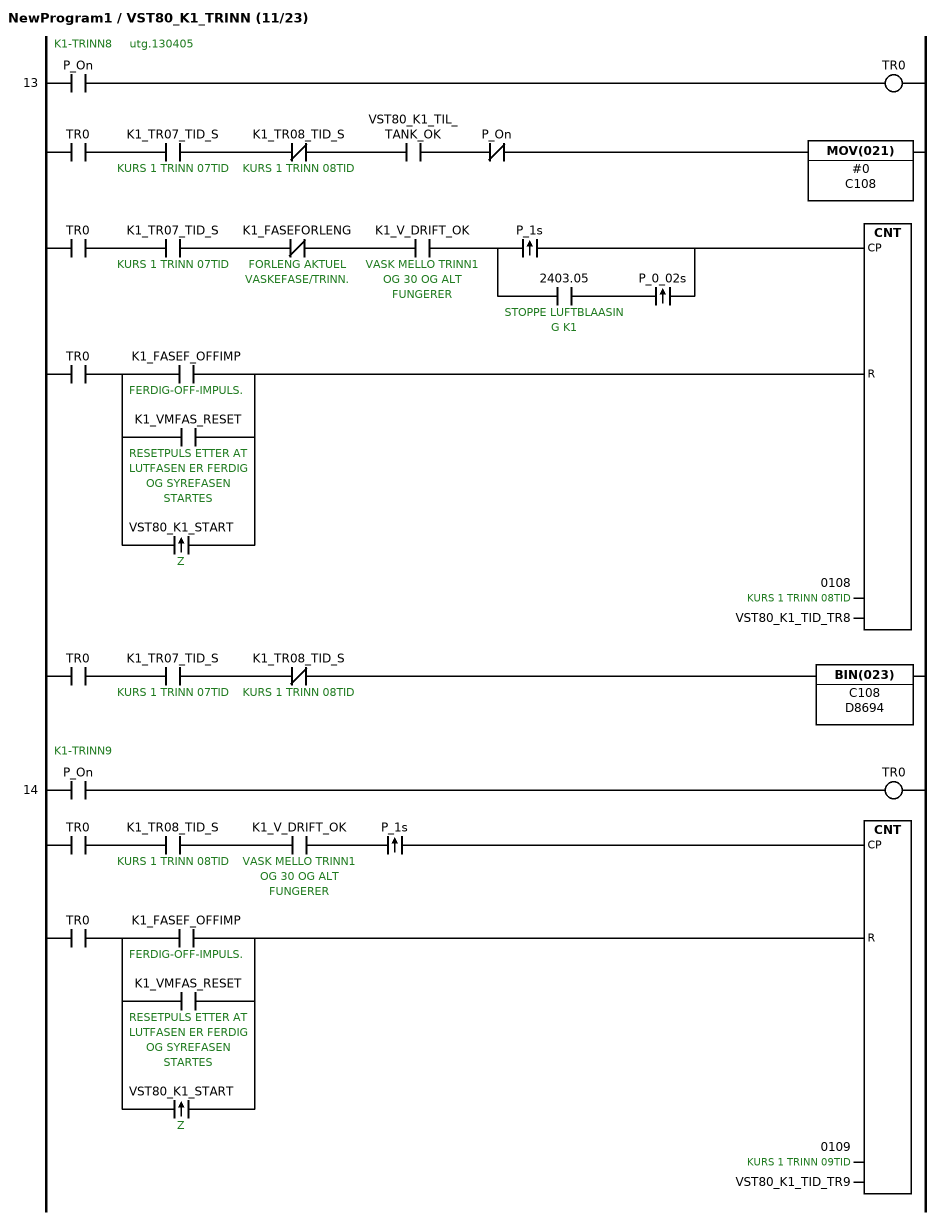
; [picture p96: NewProgram1 / VST80_K1_TRINN, rungs 13-14]
; rung 13: K1-TRINN8     utg.130405
LD P_On
OUT TR0
AND K1_TR07_TID_S  ; KURS 1 TRINN 07TID
ANDNOT K1_TR08_TID_S  ; KURS 1 TRINN 08TID
AND VST80_K1_TIL_TANK_OK
ANDNOT P_On
MOV(021) #0 C108
LD TR0
AND K1_TR07_TID_S  ; KURS 1 TRINN 07TID
ANDNOT K1_FASEFORLENG  ; FORLENG AKTUEL VASKEFASE/TRINN.
AND K1_V_DRIFT_OK  ; VASK MELLO TRINN1 OG 30 OG ALT FUNGERER
@LD P_1s
LD 2403.05  ; STOPPE LUFTBLAASING K1
@AND P_0_02s
ORLD
ANDLD
LD TR0
LD K1_FASEF_OFFIMP  ; FERDIG-OFF-IMPULS.
OR K1_VMFAS_RESET  ; RESETPULS ETTER AT LUTFASEN ER FERDIG OG SYREFASEN STARTES
@OR VST80_K1_START  ; Z
ANDLD
CNT 0108 VST80_K1_TID_TR8  ; KURS 1 TRINN 08TID
LD TR0
AND K1_TR07_TID_S  ; KURS 1 TRINN 07TID
ANDNOT K1_TR08_TID_S  ; KURS 1 TRINN 08TID
BIN(023) C108 D8694
; rung 14: K1-TRINN9
LD P_On
OUT TR0
AND K1_TR08_TID_S  ; KURS 1 TRINN 08TID
AND K1_V_DRIFT_OK  ; VASK MELLO TRINN1 OG 30 OG ALT FUNGERER
@AND P_1s
LD TR0
LD K1_FASEF_OFFIMP  ; FERDIG-OFF-IMPULS.
OR K1_VMFAS_RESET  ; RESETPULS ETTER AT LUTFASEN ER FERDIG OG SYREFASEN STARTES
@OR VST80_K1_START  ; Z
ANDLD
CNT 0109 VST80_K1_TID_TR9  ; KURS 1 TRINN 09TID

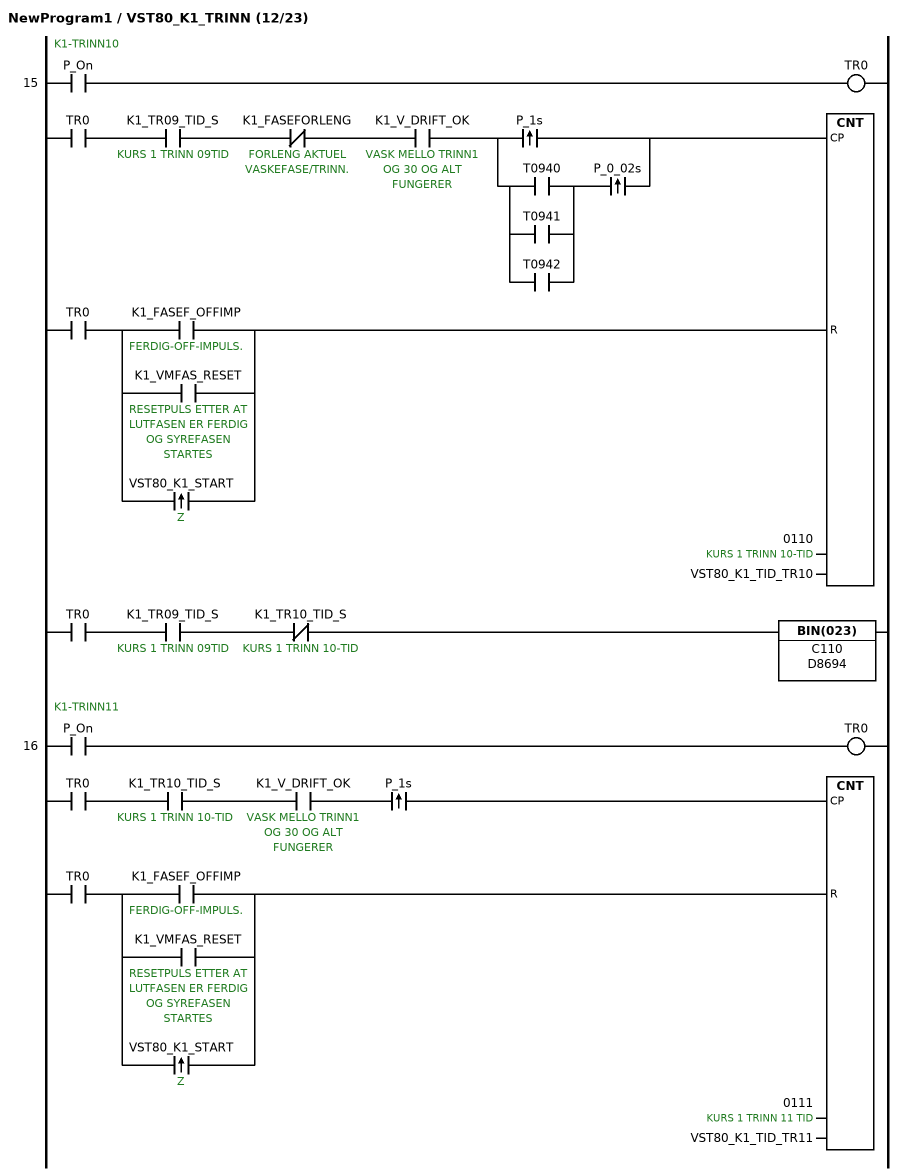
; rung 15: K1-TRINN10
LD P_On
OUT TR0
AND K1_TR09_TID_S  ; KURS 1 TRINN 09TID
ANDNOT K1_FASEFORLENG  ; FORLENG AKTUEL VASKEFASE/TRINN.
AND K1_V_DRIFT_OK  ; VASK MELLO TRINN1 OG 30 OG ALT FUNGERER
@LD P_1s
LD T0940
OR T0941
OR T0942
@AND P_0_02s
ORLD
ANDLD
LD TR0
LD K1_FASEF_OFFIMP  ; FERDIG-OFF-IMPULS.
OR K1_VMFAS_RESET  ; RESETPULS ETTER AT LUTFASEN ER FERDIG OG SYREFASEN STARTES
@OR VST80_K1_START  ; Z
ANDLD
CNT 0110 VST80_K1_TID_TR10  ; KURS 1 TRINN 10-TID
LD TR0
AND K1_TR09_TID_S  ; KURS 1 TRINN 09TID
ANDNOT K1_TR10_TID_S  ; KURS 1 TRINN 10-TID
BIN(023) C110 D8694
; rung 16: K1-TRINN11
LD P_On
OUT TR0
AND K1_TR10_TID_S  ; KURS 1 TRINN 10-TID
AND K1_V_DRIFT_OK  ; VASK MELLO TRINN1 OG 30 OG ALT FUNGERER
@AND P_1s
LD TR0
LD K1_FASEF_OFFIMP  ; FERDIG-OFF-IMPULS.
OR K1_VMFAS_RESET  ; RESETPULS ETTER AT LUTFASEN ER FERDIG OG SYREFASEN STARTES
@OR VST80_K1_START  ; Z
ANDLD
CNT 0111 VST80_K1_TID_TR11  ; KURS 1 TRINN 11 TID

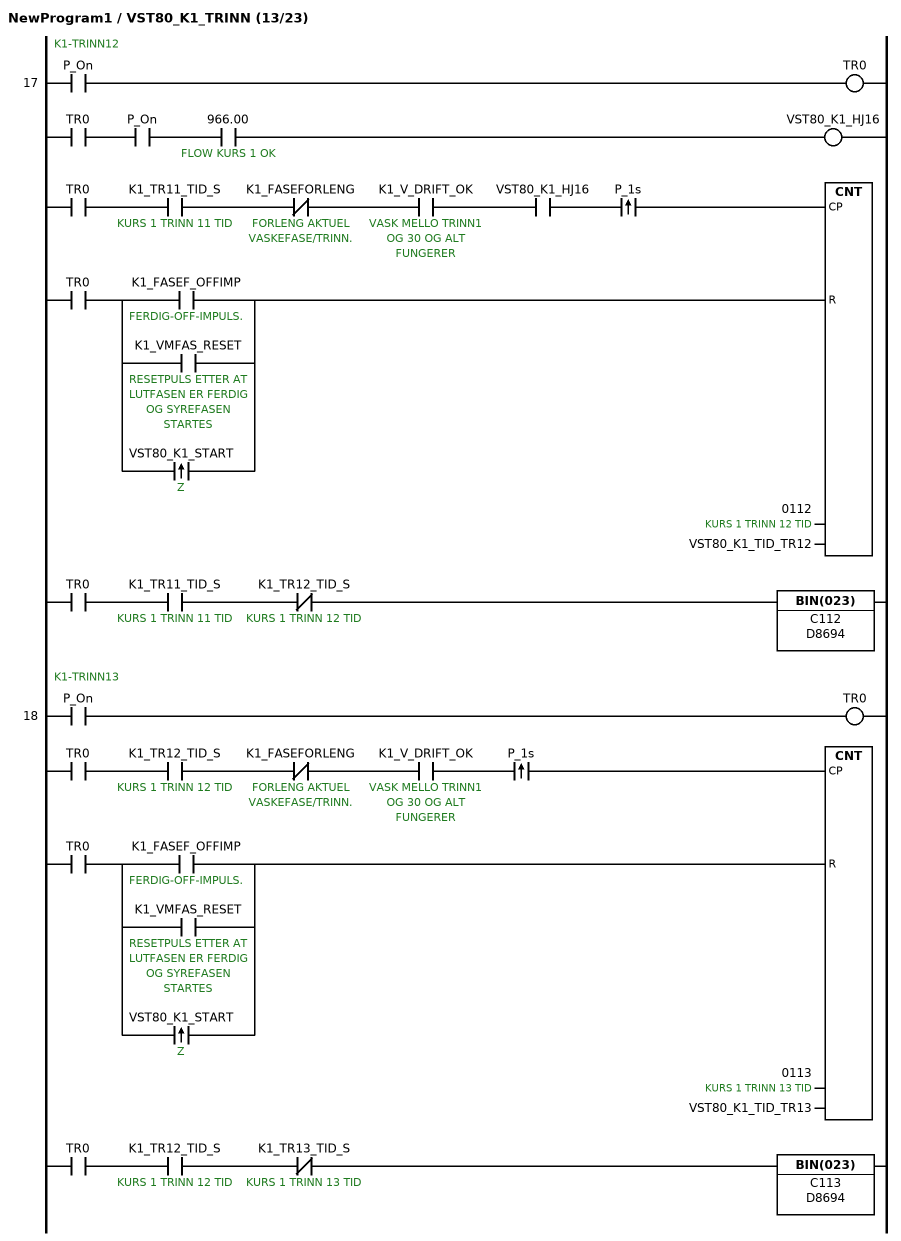
; rung 17: K1-TRINN12
LD P_On
OUT TR0
AND P_On
AND 966.00  ; FLOW KURS 1 OK
OUT VST80_K1_HJ16
LD TR0
AND K1_TR11_TID_S  ; KURS 1 TRINN 11 TID
ANDNOT K1_FASEFORLENG  ; FORLENG AKTUEL VASKEFASE/TRINN.
AND K1_V_DRIFT_OK  ; VASK MELLO TRINN1 OG 30 OG ALT FUNGERER
AND VST80_K1_HJ16
@AND P_1s
LD TR0
LD K1_FASEF_OFFIMP  ; FERDIG-OFF-IMPULS.
OR K1_VMFAS_RESET  ; RESETPULS ETTER AT LUTFASEN ER FERDIG OG SYREFASEN STARTES
@OR VST80_K1_START  ; Z
ANDLD
CNT 0112 VST80_K1_TID_TR12  ; KURS 1 TRINN 12 TID
LD TR0
AND K1_TR11_TID_S  ; KURS 1 TRINN 11 TID
ANDNOT K1_TR12_TID_S  ; KURS 1 TRINN 12 TID
BIN(023) C112 D8694
; rung 18: K1-TRINN13
LD P_On
OUT TR0
AND K1_TR12_TID_S  ; KURS 1 TRINN 12 TID
ANDNOT K1_FASEFORLENG  ; FORLENG AKTUEL VASKEFASE/TRINN.
AND K1_V_DRIFT_OK  ; VASK MELLO TRINN1 OG 30 OG ALT FUNGERER
@AND P_1s
LD TR0
LD K1_FASEF_OFFIMP  ; FERDIG-OFF-IMPULS.
OR K1_VMFAS_RESET  ; RESETPULS ETTER AT LUTFASEN ER FERDIG OG SYREFASEN STARTES
@OR VST80_K1_START  ; Z
ANDLD
CNT 0113 VST80_K1_TID_TR13  ; KURS 1 TRINN 13 TID
LD TR0
AND K1_TR12_TID_S  ; KURS 1 TRINN 12 TID
ANDNOT K1_TR13_TID_S  ; KURS 1 TRINN 13 TID
BIN(023) C113 D8694

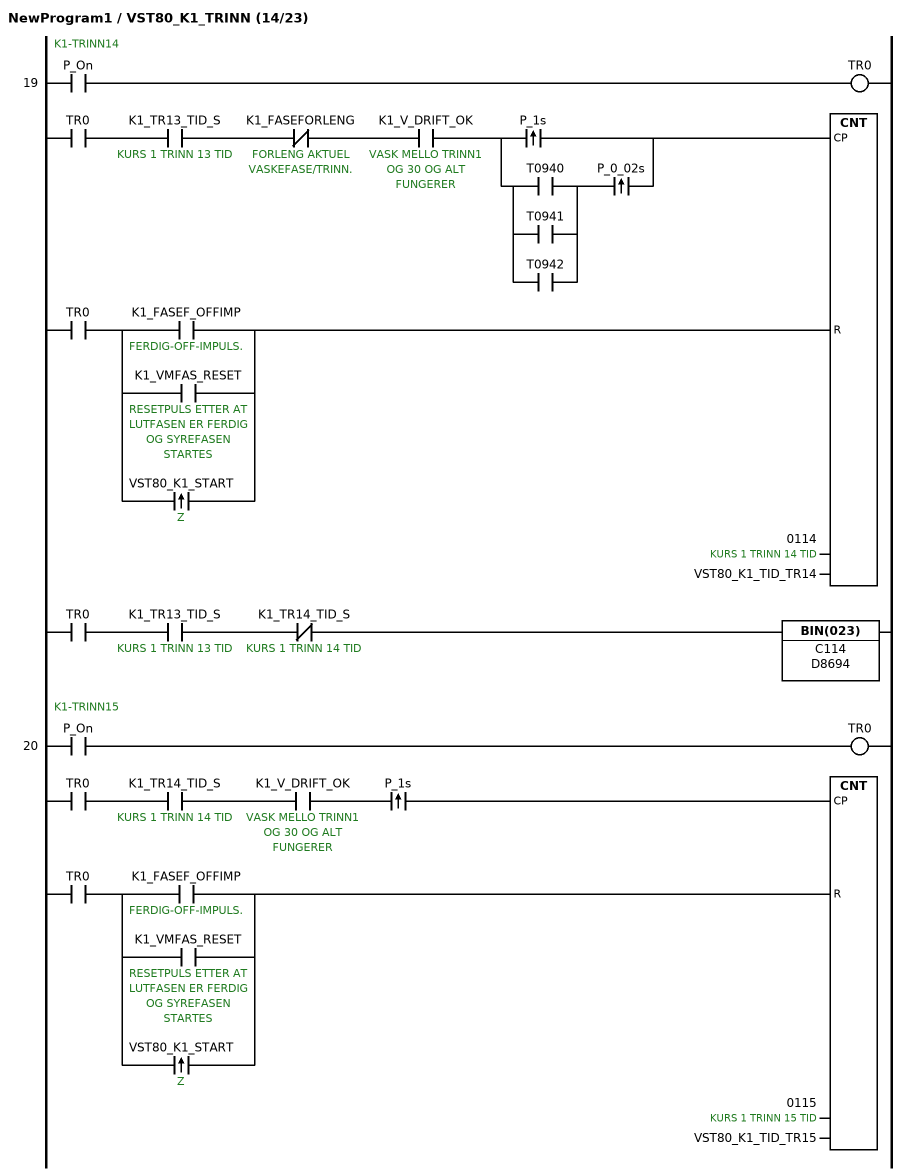
; rung 19: K1-TRINN14
LD P_On
OUT TR0
AND K1_TR13_TID_S  ; KURS 1 TRINN 13 TID
ANDNOT K1_FASEFORLENG  ; FORLENG AKTUEL VASKEFASE/TRINN.
AND K1_V_DRIFT_OK  ; VASK MELLO TRINN1 OG 30 OG ALT FUNGERER
@LD P_1s
LD T0940
OR T0941
OR T0942
@AND P_0_02s
ORLD
ANDLD
LD TR0
LD K1_FASEF_OFFIMP  ; FERDIG-OFF-IMPULS.
OR K1_VMFAS_RESET  ; RESETPULS ETTER AT LUTFASEN ER FERDIG OG SYREFASEN STARTES
@OR VST80_K1_START  ; Z
ANDLD
CNT 0114 VST80_K1_TID_TR14  ; KURS 1 TRINN 14 TID
LD TR0
AND K1_TR13_TID_S  ; KURS 1 TRINN 13 TID
ANDNOT K1_TR14_TID_S  ; KURS 1 TRINN 14 TID
BIN(023) C114 D8694
; rung 20: K1-TRINN15
LD P_On
OUT TR0
AND K1_TR14_TID_S  ; KURS 1 TRINN 14 TID
AND K1_V_DRIFT_OK  ; VASK MELLO TRINN1 OG 30 OG ALT FUNGERER
@AND P_1s
LD TR0
LD K1_FASEF_OFFIMP  ; FERDIG-OFF-IMPULS.
OR K1_VMFAS_RESET  ; RESETPULS ETTER AT LUTFASEN ER FERDIG OG SYREFASEN STARTES
@OR VST80_K1_START  ; Z
ANDLD
CNT 0115 VST80_K1_TID_TR15  ; KURS 1 TRINN 15 TID

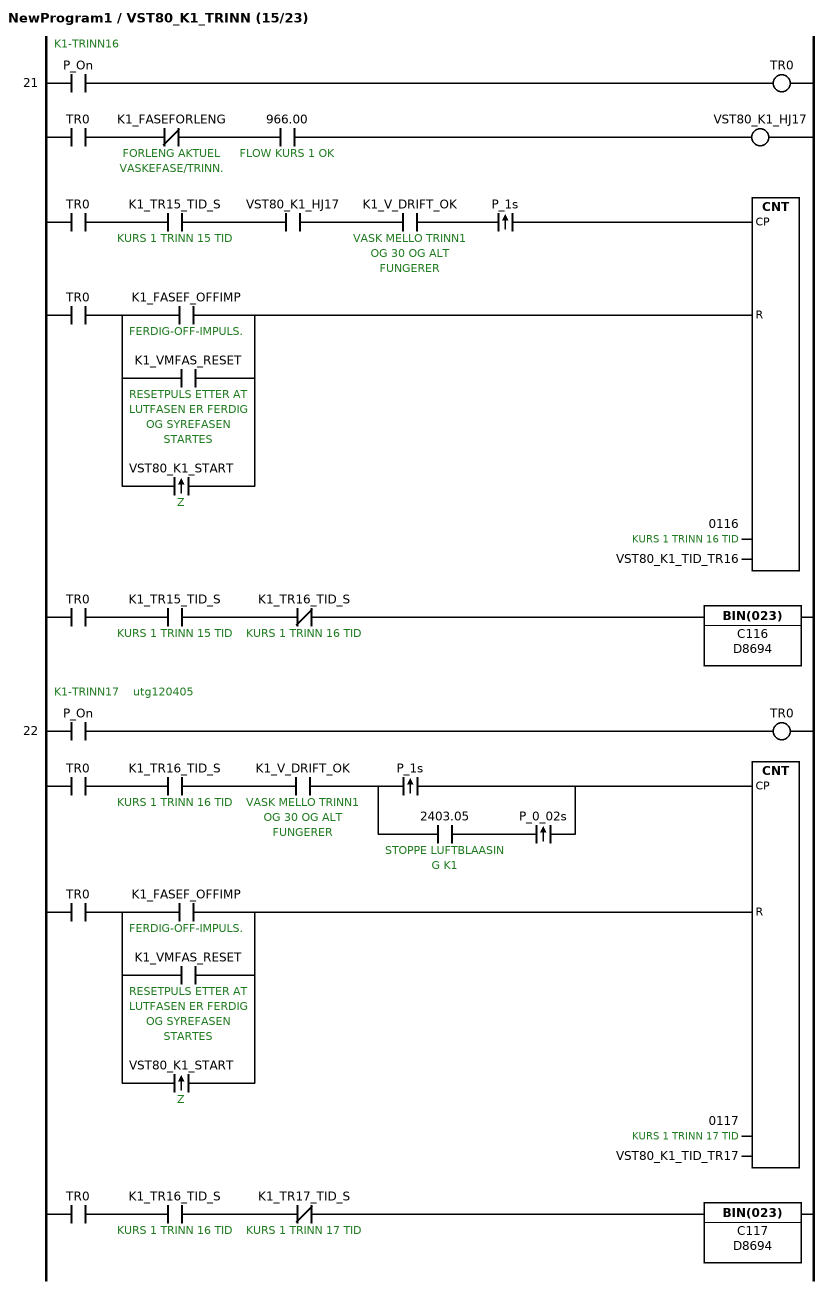
; rung 21: K1-TRINN16
LD P_On
OUT TR0
ANDNOT K1_FASEFORLENG  ; FORLENG AKTUEL VASKEFASE/TRINN.
AND 966.00  ; FLOW KURS 1 OK
OUT VST80_K1_HJ17
LD TR0
AND K1_TR15_TID_S  ; KURS 1 TRINN 15 TID
AND VST80_K1_HJ17
AND K1_V_DRIFT_OK  ; VASK MELLO TRINN1 OG 30 OG ALT FUNGERER
@AND P_1s
LD TR0
LD K1_FASEF_OFFIMP  ; FERDIG-OFF-IMPULS.
OR K1_VMFAS_RESET  ; RESETPULS ETTER AT LUTFASEN ER FERDIG OG SYREFASEN STARTES
@OR VST80_K1_START  ; Z
ANDLD
CNT 0116 VST80_K1_TID_TR16  ; KURS 1 TRINN 16 TID
LD TR0
AND K1_TR15_TID_S  ; KURS 1 TRINN 15 TID
ANDNOT K1_TR16_TID_S  ; KURS 1 TRINN 16 TID
BIN(023) C116 D8694
; rung 22: K1-TRINN17    utg120405
LD P_On
OUT TR0
AND K1_TR16_TID_S  ; KURS 1 TRINN 16 TID
AND K1_V_DRIFT_OK  ; VASK MELLO TRINN1 OG 30 OG ALT FUNGERER
@LD P_1s
LD 2403.05  ; STOPPE LUFTBLAASING K1
@AND P_0_02s
ORLD
ANDLD
LD TR0
LD K1_FASEF_OFFIMP  ; FERDIG-OFF-IMPULS.
OR K1_VMFAS_RESET  ; RESETPULS ETTER AT LUTFASEN ER FERDIG OG SYREFASEN STARTES
@OR VST80_K1_START  ; Z
ANDLD
CNT 0117 VST80_K1_TID_TR17  ; KURS 1 TRINN 17 TID
LD TR0
AND K1_TR16_TID_S  ; KURS 1 TRINN 16 TID
ANDNOT K1_TR17_TID_S  ; KURS 1 TRINN 17 TID
BIN(023) C117 D8694

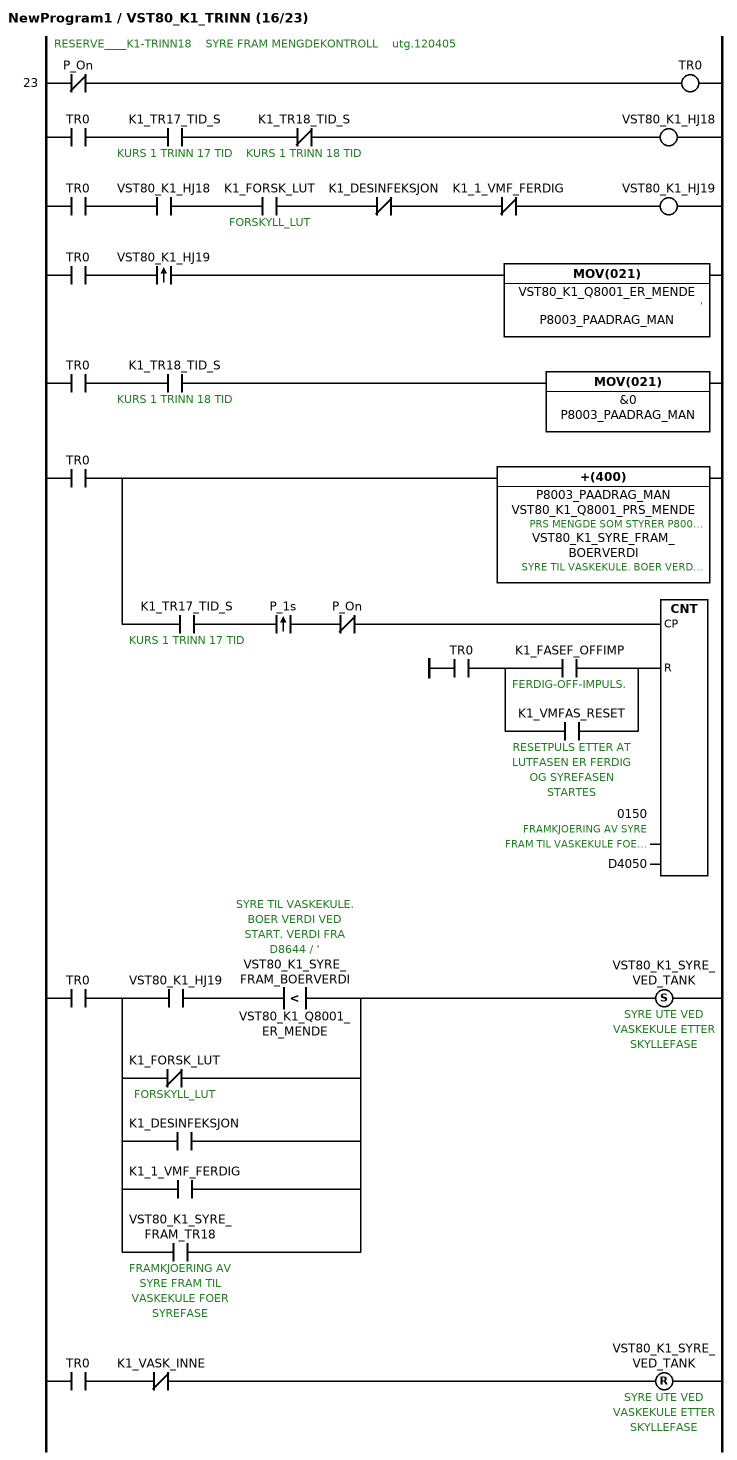
; rung 23: RESERVE____K1-TRINN18    SYRE FRAM MENGDEKONTROLL    utg.120405
LDNOT P_On
OUT TR0
AND K1_TR17_TID_S  ; KURS 1 TRINN 17 TID
ANDNOT K1_TR18_TID_S  ; KURS 1 TRINN 18 TID
OUT VST80_K1_HJ18
LD TR0
AND VST80_K1_HJ18
AND K1_FORSK_LUT  ; FORSKYLL_LUT
ANDNOT K1_DESINFEKSJON
ANDNOT K1_1_VMF_FERDIG
OUT VST80_K1_HJ19
LD TR0
@AND VST80_K1_HJ19
MOV(021) VST80_K1_Q8001_ER_MENDE P8003_PAADRAG_MAN  ; '
LD TR0
AND K1_TR18_TID_S  ; KURS 1 TRINN 18 TID
MOV(021) &0 P8003_PAADRAG_MAN
LD TR0
+(400) P8003_PAADRAG_MAN VST80_K1_Q8001_PRS_MENDE VST80_K1_SYRE_FRAM_BOERVERDI  ; PRS MENGDE SOM STYRER P8001 VED FASESKIFTE, SYRE TIL VASKEKULE. BOER VERDI VED START. VERDI FRA D8644
AND K1_TR17_TID_S  ; KURS 1 TRINN 17 TID
@AND P_1s
ANDNOT P_On
LD TR0
LD K1_FASEF_OFFIMP  ; FERDIG-OFF-IMPULS.
OR K1_VMFAS_RESET  ; RESETPULS ETTER AT LUTFASEN ER FERDIG OG SYREFASEN STARTES
ANDLD
CNT 0150 D4050  ; FRAMKJOERING AV SYRE FRAM TIL VASKEKULE FOER SYREFASE
LD TR0
LD VST80_K1_HJ19
AND<(310) VST80_K1_SYRE_FRAM_BOERVERDI VST80_K1_Q8001_ER_MENDE  ; SYRE TIL VASKEKULE. BOER VERDI VED START. VERDI FRA D8644, '
ORNOT K1_FORSK_LUT  ; FORSKYLL_LUT
OR K1_DESINFEKSJON
OR K1_1_VMF_FERDIG
OR VST80_K1_SYRE_FRAM_TR18  ; FRAMKJOERING AV SYRE FRAM TIL VASKEKULE FOER SYREFASE
ANDLD
SET VST80_K1_SYRE_VED_TANK  ; SYRE UTE VED VASKEKULE ETTER SKYLLEFASE
LD TR0
ANDNOT K1_VASK_INNE
RSET VST80_K1_SYRE_VED_TANK  ; SYRE UTE VED VASKEKULE ETTER SKYLLEFASE

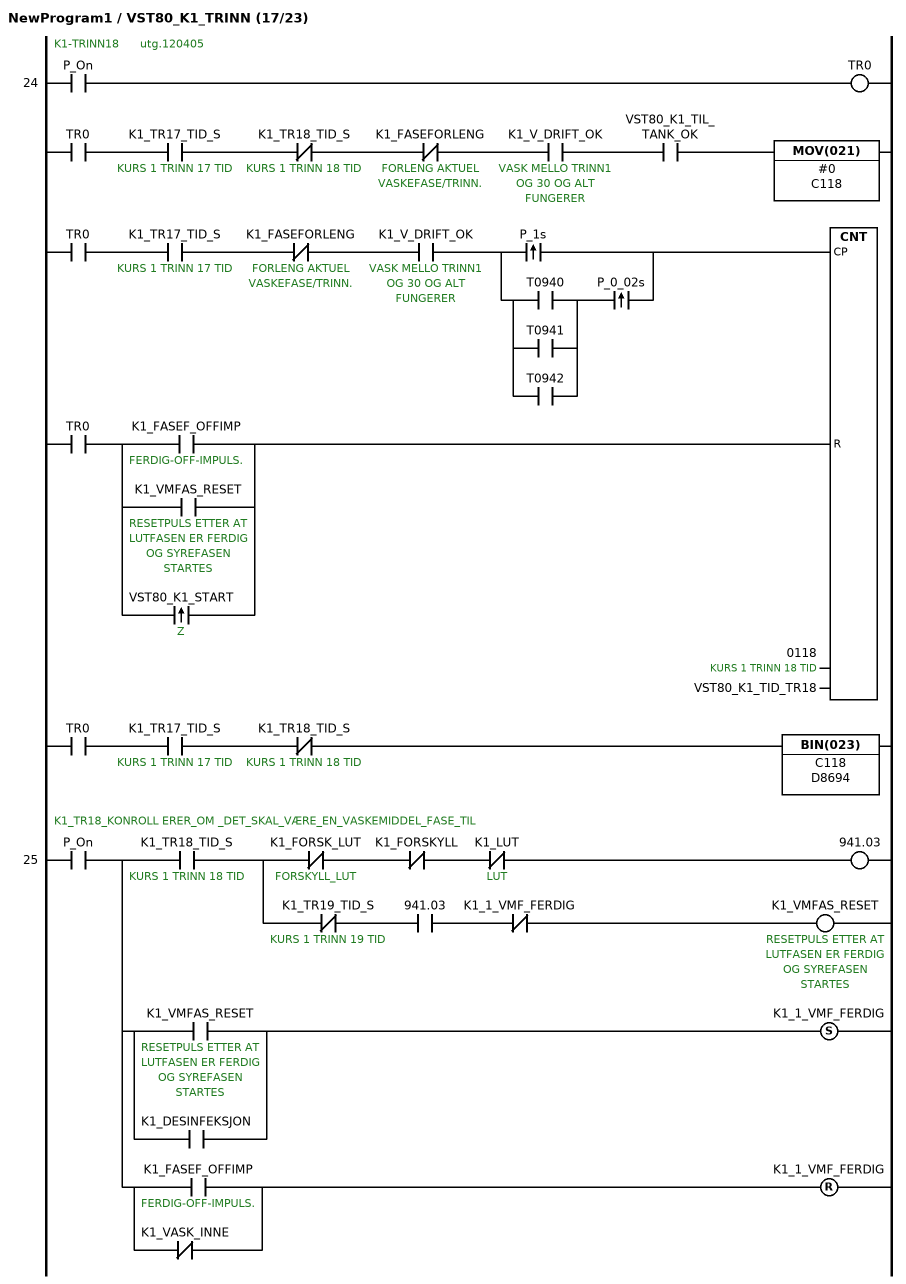
; rung 24: K1-TRINN18      utg.120405
LD P_On
OUT TR0
AND K1_TR17_TID_S  ; KURS 1 TRINN 17 TID
ANDNOT K1_TR18_TID_S  ; KURS 1 TRINN 18 TID
ANDNOT K1_FASEFORLENG  ; FORLENG AKTUEL VASKEFASE/TRINN.
AND K1_V_DRIFT_OK  ; VASK MELLO TRINN1 OG 30 OG ALT FUNGERER
AND VST80_K1_TIL_TANK_OK
MOV(021) #0 C118
LD TR0
AND K1_TR17_TID_S  ; KURS 1 TRINN 17 TID
ANDNOT K1_FASEFORLENG  ; FORLENG AKTUEL VASKEFASE/TRINN.
AND K1_V_DRIFT_OK  ; VASK MELLO TRINN1 OG 30 OG ALT FUNGERER
@LD P_1s
LD T0940
OR T0941
OR T0942
@AND P_0_02s
ORLD
ANDLD
LD TR0
LD K1_FASEF_OFFIMP  ; FERDIG-OFF-IMPULS.
OR K1_VMFAS_RESET  ; RESETPULS ETTER AT LUTFASEN ER FERDIG OG SYREFASEN STARTES
@OR VST80_K1_START  ; Z
ANDLD
CNT 0118 VST80_K1_TID_TR18  ; KURS 1 TRINN 18 TID
LD TR0
AND K1_TR17_TID_S  ; KURS 1 TRINN 17 TID
ANDNOT K1_TR18_TID_S  ; KURS 1 TRINN 18 TID
BIN(023) C118 D8694
; rung 25: K1_TR18_KONROLL ERER_OM_DET_SKAL_VÆRE_EN_VASKEMIDDEL_FASE_TIL
LD P_On
OUT TR0
AND K1_TR18_TID_S  ; KURS 1 TRINN 18 TID
OUT TR1
ANDNOT K1_FORSK_LUT  ; FORSKYLL_LUT
ANDNOT K1_FORSKYLL
ANDNOT K1_LUT  ; LUT
OUT 941.03
LD TR1
ANDNOT K1_TR19_TID_S  ; KURS 1 TRINN 19 TID
AND 941.03
ANDNOT K1_1_VMF_FERDIG
OUT K1_VMFAS_RESET  ; RESETPULS ETTER AT LUTFASEN ER FERDIG OG SYREFASEN STARTES
LD TR0
LD K1_VMFAS_RESET  ; RESETPULS ETTER AT LUTFASEN ER FERDIG OG SYREFASEN STARTES
OR K1_DESINFEKSJON
ANDLD
SET K1_1_VMF_FERDIG
LD TR0
LD K1_FASEF_OFFIMP  ; FERDIG-OFF-IMPULS.
ORNOT K1_VASK_INNE
ANDLD
RSET K1_1_VMF_FERDIG

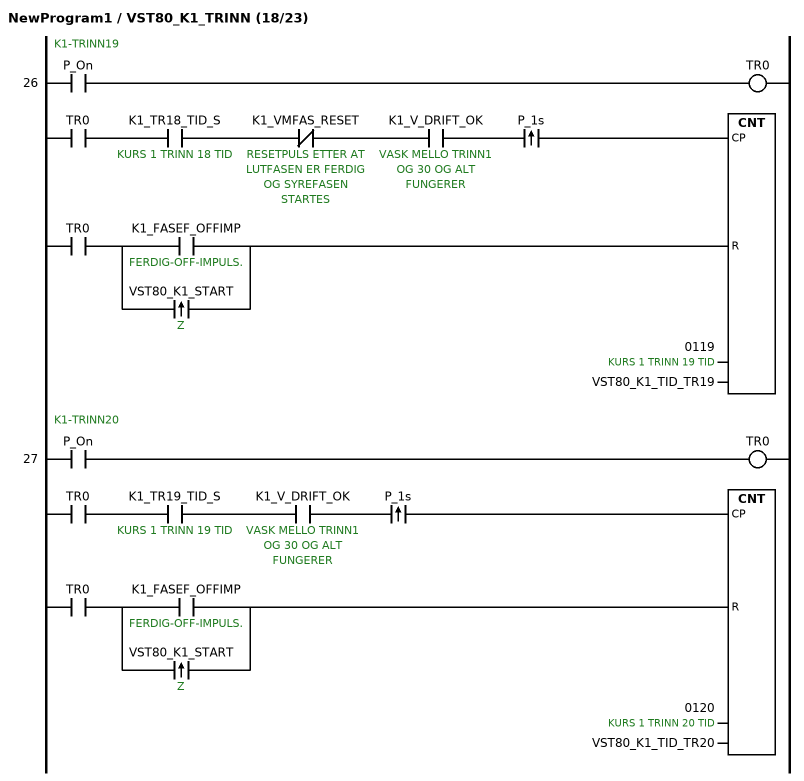
; rung 26: K1-TRINN19
LD P_On
OUT TR0
AND K1_TR18_TID_S  ; KURS 1 TRINN 18 TID
ANDNOT K1_VMFAS_RESET  ; RESETPULS ETTER AT LUTFASEN ER FERDIG OG SYREFASEN STARTES
AND K1_V_DRIFT_OK  ; VASK MELLO TRINN1 OG 30 OG ALT FUNGERER
@AND P_1s
LD TR0
LD K1_FASEF_OFFIMP  ; FERDIG-OFF-IMPULS.
@OR VST80_K1_START  ; Z
ANDLD
CNT 0119 VST80_K1_TID_TR19  ; KURS 1 TRINN 19 TID
; rung 27: K1-TRINN20
LD P_On
OUT TR0
AND K1_TR19_TID_S  ; KURS 1 TRINN 19 TID
AND K1_V_DRIFT_OK  ; VASK MELLO TRINN1 OG 30 OG ALT FUNGERER
@AND P_1s
LD TR0
LD K1_FASEF_OFFIMP  ; FERDIG-OFF-IMPULS.
@OR VST80_K1_START  ; Z
ANDLD
CNT 0120 VST80_K1_TID_TR20  ; KURS 1 TRINN 20 TID

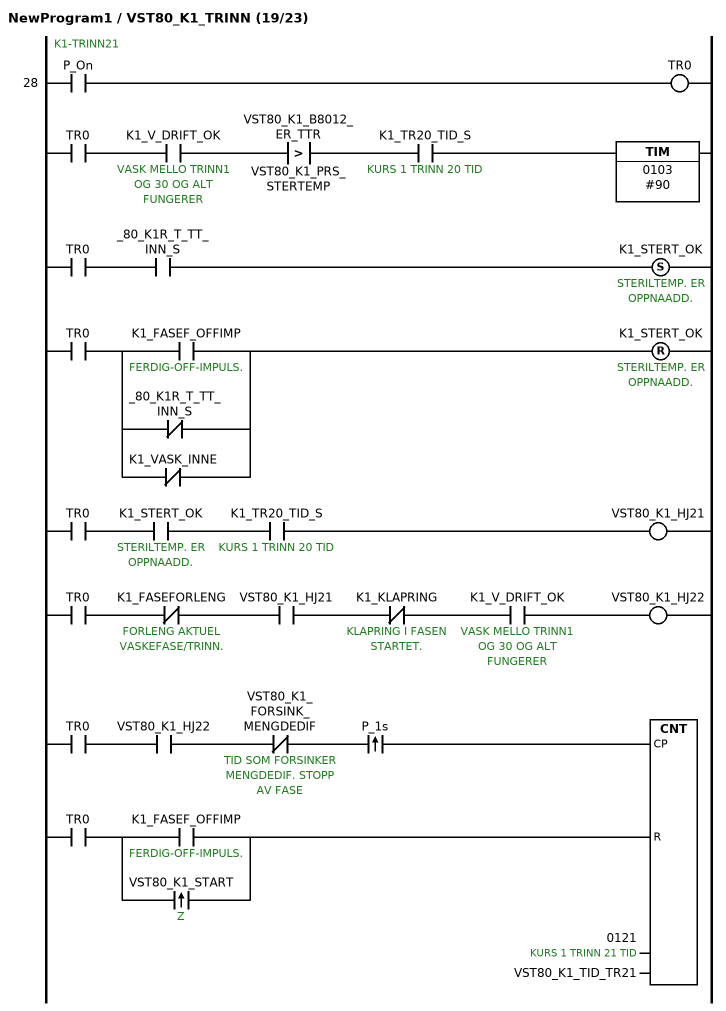
; rung 28: K1-TRINN21
LD P_On
OUT TR0
AND K1_V_DRIFT_OK  ; VASK MELLO TRINN1 OG 30 OG ALT FUNGERER
AND>(320) VST80_K1_B8012_ER_TTR VST80_K1_PRS_STERTEMP
AND K1_TR20_TID_S  ; KURS 1 TRINN 20 TID
TIM 0103 #90
LD TR0
AND _80_K1R_T_TT_INN_S
SET K1_STERT_OK  ; STERILTEMP. ER OPPNAADD.
LD TR0
LD K1_FASEF_OFFIMP  ; FERDIG-OFF-IMPULS.
ORNOT _80_K1R_T_TT_INN_S
ORNOT K1_VASK_INNE
ANDLD
RSET K1_STERT_OK  ; STERILTEMP. ER OPPNAADD.
LD TR0
AND K1_STERT_OK  ; STERILTEMP. ER OPPNAADD.
AND K1_TR20_TID_S  ; KURS 1 TRINN 20 TID
OUT VST80_K1_HJ21
LD TR0
ANDNOT K1_FASEFORLENG  ; FORLENG AKTUEL VASKEFASE/TRINN.
AND VST80_K1_HJ21
ANDNOT K1_KLAPRING  ; KLAPRING I FASEN STARTET.
AND K1_V_DRIFT_OK  ; VASK MELLO TRINN1 OG 30 OG ALT FUNGERER
OUT VST80_K1_HJ22
LD TR0
AND VST80_K1_HJ22
ANDNOT VST80_K1_FORSINK_MENGDEDIF  ; TID SOM FORSINKER MENGDEDIF. STOPP AV FASE
@AND P_1s
LD TR0
LD K1_FASEF_OFFIMP  ; FERDIG-OFF-IMPULS.
@OR VST80_K1_START  ; Z
ANDLD
CNT 0121 VST80_K1_TID_TR21  ; KURS 1 TRINN 21 TID

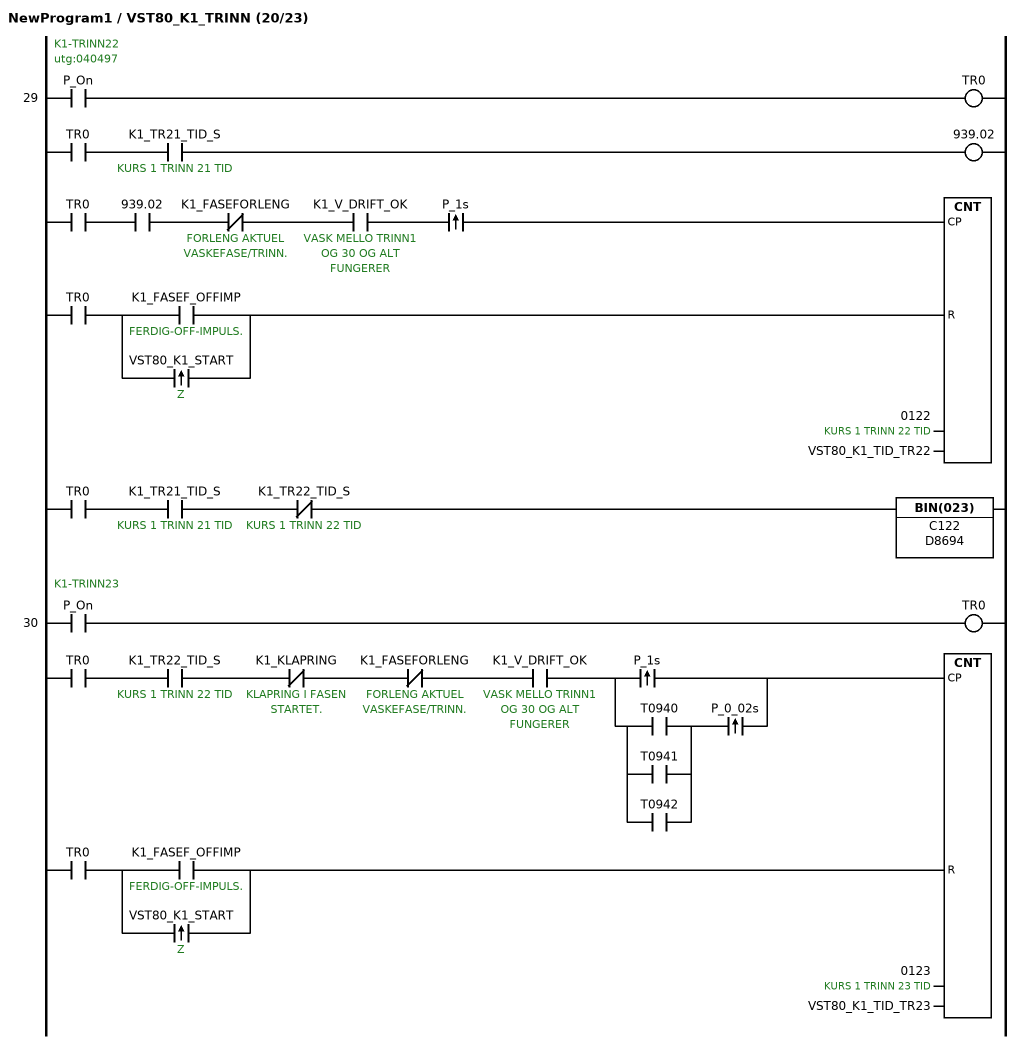
; rung 29: K1-TRINN22 / utg:040497
LD P_On
OUT TR0
AND K1_TR21_TID_S  ; KURS 1 TRINN 21 TID
OUT 939.02
LD TR0
AND 939.02
ANDNOT K1_FASEFORLENG  ; FORLENG AKTUEL VASKEFASE/TRINN.
AND K1_V_DRIFT_OK  ; VASK MELLO TRINN1 OG 30 OG ALT FUNGERER
@AND P_1s
LD TR0
LD K1_FASEF_OFFIMP  ; FERDIG-OFF-IMPULS.
@OR VST80_K1_START  ; Z
ANDLD
CNT 0122 VST80_K1_TID_TR22  ; KURS 1 TRINN 22 TID
LD TR0
AND K1_TR21_TID_S  ; KURS 1 TRINN 21 TID
ANDNOT K1_TR22_TID_S  ; KURS 1 TRINN 22 TID
BIN(023) C122 D8694
; rung 30: K1-TRINN23
LD P_On
OUT TR0
AND K1_TR22_TID_S  ; KURS 1 TRINN 22 TID
ANDNOT K1_KLAPRING  ; KLAPRING I FASEN STARTET.
ANDNOT K1_FASEFORLENG  ; FORLENG AKTUEL VASKEFASE/TRINN.
AND K1_V_DRIFT_OK  ; VASK MELLO TRINN1 OG 30 OG ALT FUNGERER
@LD P_1s
LD T0940
OR T0941
OR T0942
@AND P_0_02s
ORLD
ANDLD
LD TR0
LD K1_FASEF_OFFIMP  ; FERDIG-OFF-IMPULS.
@OR VST80_K1_START  ; Z
ANDLD
CNT 0123 VST80_K1_TID_TR23  ; KURS 1 TRINN 23 TID

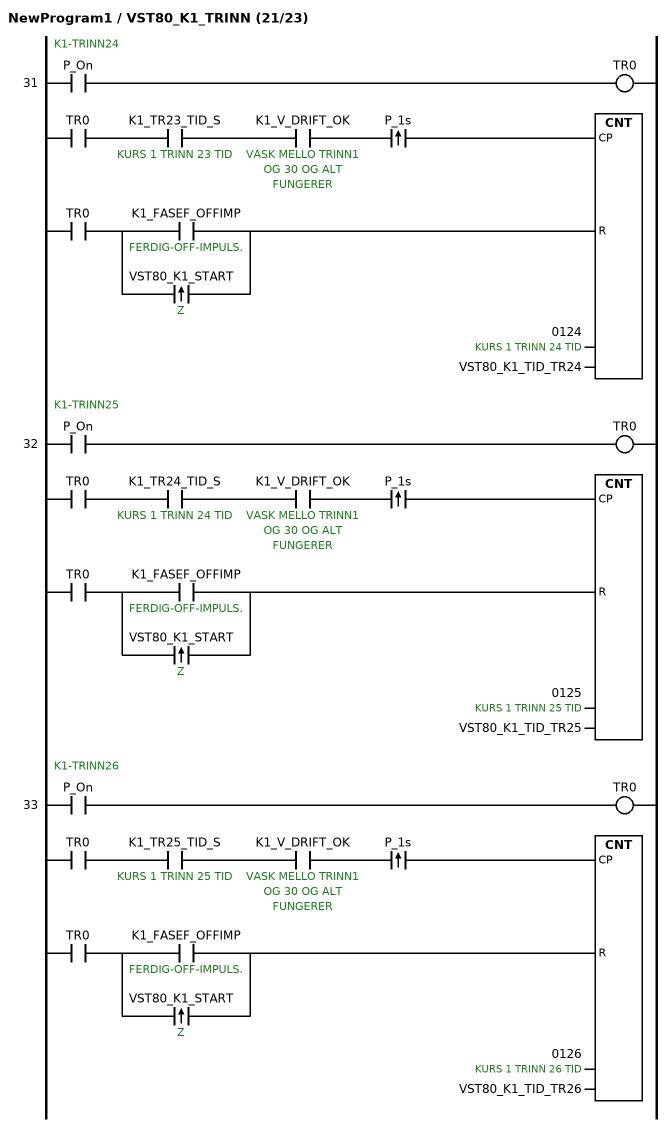
; rung 31: K1-TRINN24
LD P_On
OUT TR0
AND K1_TR23_TID_S  ; KURS 1 TRINN 23 TID
AND K1_V_DRIFT_OK  ; VASK MELLO TRINN1 OG 30 OG ALT FUNGERER
@AND P_1s
LD TR0
LD K1_FASEF_OFFIMP  ; FERDIG-OFF-IMPULS.
@OR VST80_K1_START  ; Z
ANDLD
CNT 0124 VST80_K1_TID_TR24  ; KURS 1 TRINN 24 TID
; rung 32: K1-TRINN25
LD P_On
OUT TR0
AND K1_TR24_TID_S  ; KURS 1 TRINN 24 TID
AND K1_V_DRIFT_OK  ; VASK MELLO TRINN1 OG 30 OG ALT FUNGERER
@AND P_1s
LD TR0
LD K1_FASEF_OFFIMP  ; FERDIG-OFF-IMPULS.
@OR VST80_K1_START  ; Z
ANDLD
CNT 0125 VST80_K1_TID_TR25  ; KURS 1 TRINN 25 TID
; rung 33: K1-TRINN26
LD P_On
OUT TR0
AND K1_TR25_TID_S  ; KURS 1 TRINN 25 TID
AND K1_V_DRIFT_OK  ; VASK MELLO TRINN1 OG 30 OG ALT FUNGERER
@AND P_1s
LD TR0
LD K1_FASEF_OFFIMP  ; FERDIG-OFF-IMPULS.
@OR VST80_K1_START  ; Z
ANDLD
CNT 0126 VST80_K1_TID_TR26  ; KURS 1 TRINN 26 TID

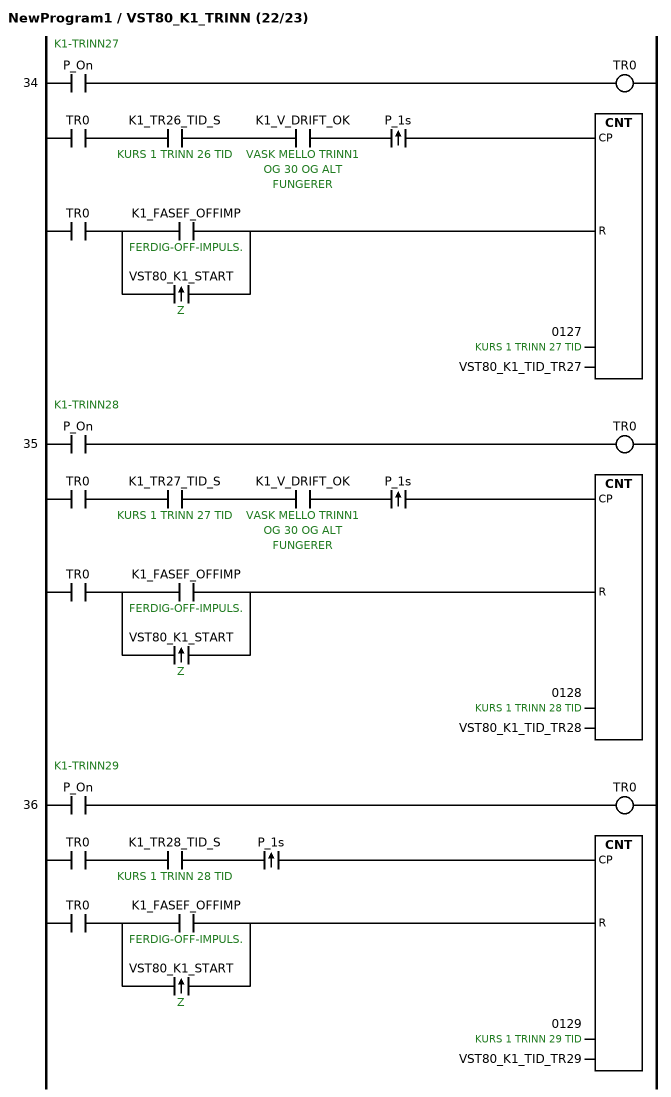
; rung 34: K1-TRINN27
LD P_On
OUT TR0
AND K1_TR26_TID_S  ; KURS 1 TRINN 26 TID
AND K1_V_DRIFT_OK  ; VASK MELLO TRINN1 OG 30 OG ALT FUNGERER
@AND P_1s
LD TR0
LD K1_FASEF_OFFIMP  ; FERDIG-OFF-IMPULS.
@OR VST80_K1_START  ; Z
ANDLD
CNT 0127 VST80_K1_TID_TR27  ; KURS 1 TRINN 27 TID
; rung 35: K1-TRINN28
LD P_On
OUT TR0
AND K1_TR27_TID_S  ; KURS 1 TRINN 27 TID
AND K1_V_DRIFT_OK  ; VASK MELLO TRINN1 OG 30 OG ALT FUNGERER
@AND P_1s
LD TR0
LD K1_FASEF_OFFIMP  ; FERDIG-OFF-IMPULS.
@OR VST80_K1_START  ; Z
ANDLD
CNT 0128 VST80_K1_TID_TR28  ; KURS 1 TRINN 28 TID
; rung 36: K1-TRINN29
LD P_On
OUT TR0
AND K1_TR28_TID_S  ; KURS 1 TRINN 28 TID
@AND P_1s
LD TR0
LD K1_FASEF_OFFIMP  ; FERDIG-OFF-IMPULS.
@OR VST80_K1_START  ; Z
ANDLD
CNT 0129 VST80_K1_TID_TR29  ; KURS 1 TRINN 29 TID

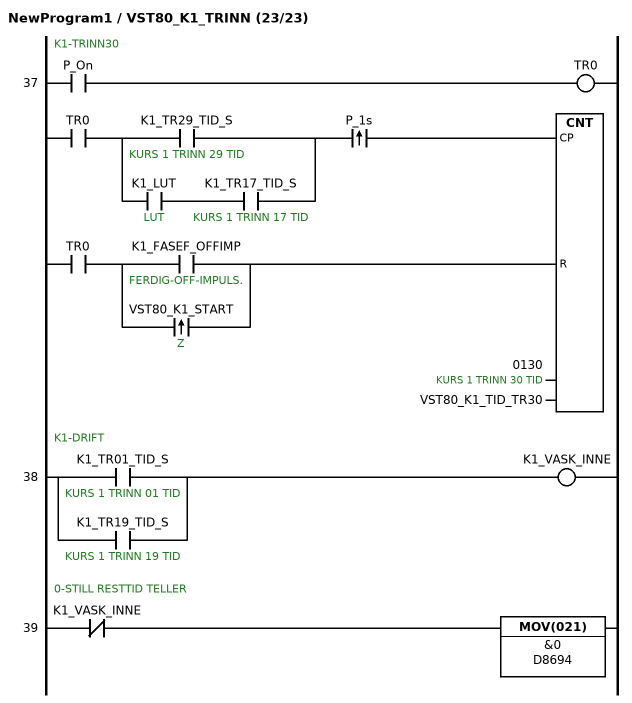
; rung 37: K1-TRINN30
LD P_On
OUT TR0
LD K1_TR29_TID_S  ; KURS 1 TRINN 29 TID
LD K1_LUT  ; LUT
AND K1_TR17_TID_S  ; KURS 1 TRINN 17 TID
ORLD
ANDLD
@AND P_1s
LD TR0
LD K1_FASEF_OFFIMP  ; FERDIG-OFF-IMPULS.
@OR VST80_K1_START  ; Z
ANDLD
CNT 0130 VST80_K1_TID_TR30  ; KURS 1 TRINN 30 TID
; rung 38: K1-DRIFT
LD K1_TR01_TID_S  ; KURS 1 TRINN 01 TID
OR K1_TR19_TID_S  ; KURS 1 TRINN 19 TID
OUT K1_VASK_INNE
; rung 39: 0-STILL RESTTID TELLER
LDNOT K1_VASK_INNE
MOV(021) &0 D8694

### Section VST_80_K1_TYPE_VASK
; KOMMANDOGIVNING FOR VALG AV TYPE VASK. / 2: DESINFEKSJON / 3: FORSKYLL

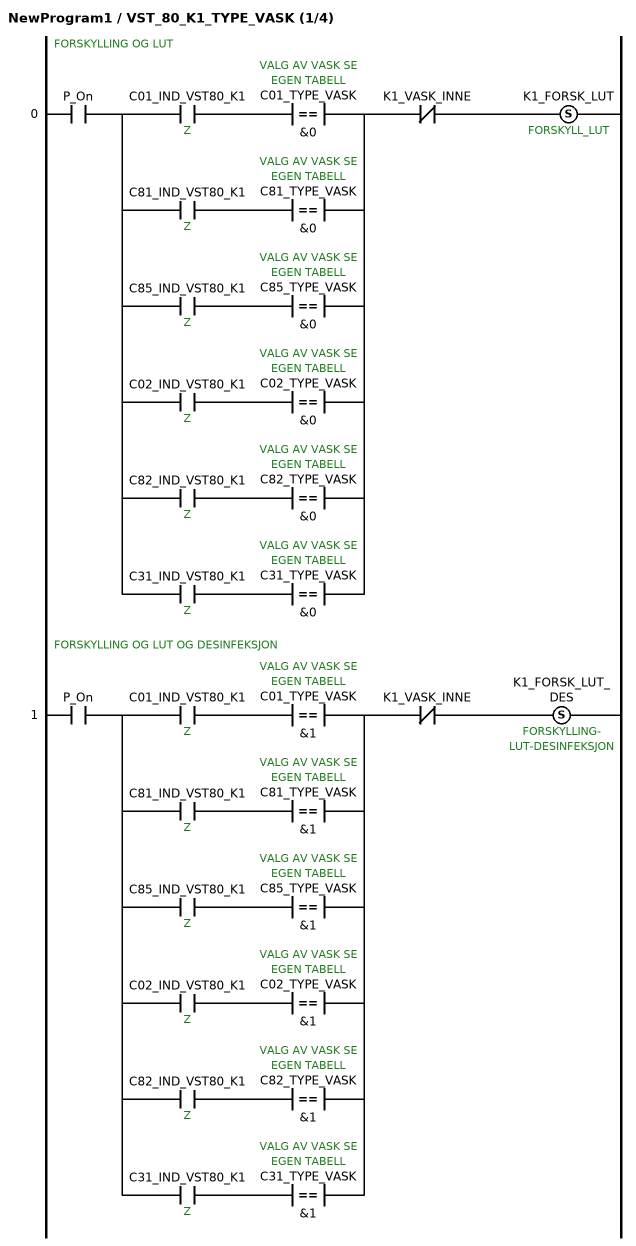
; rung 0: FORSKYLLING OG LUT
LD P_On
LD C01_IND_VST80_K1  ; Z
AND=(300) C01_TYPE_VASK &0  ; VALG AV VASK SE EGEN TABELL
LD C81_IND_VST80_K1  ; Z
AND=(300) C81_TYPE_VASK &0  ; VALG AV VASK SE EGEN TABELL
ORLD
LD C85_IND_VST80_K1  ; Z
AND=(300) C85_TYPE_VASK &0  ; VALG AV VASK SE EGEN TABELL
ORLD
LD C02_IND_VST80_K1  ; Z
AND=(300) C02_TYPE_VASK &0  ; VALG AV VASK SE EGEN TABELL
ORLD
LD C82_IND_VST80_K1  ; Z
AND=(300) C82_TYPE_VASK &0  ; VALG AV VASK SE EGEN TABELL
ORLD
LD C31_IND_VST80_K1  ; Z
AND=(300) C31_TYPE_VASK &0  ; VALG AV VASK SE EGEN TABELL
ORLD
ANDLD
ANDNOT K1_VASK_INNE
SET K1_FORSK_LUT  ; FORSKYLL_LUT
; rung 1: FORSKYLLING OG LUT OG DESINFEKSJON
LD P_On
LD C01_IND_VST80_K1  ; Z
AND=(300) C01_TYPE_VASK &1  ; VALG AV VASK SE EGEN TABELL
LD C81_IND_VST80_K1  ; Z
AND=(300) C81_TYPE_VASK &1  ; VALG AV VASK SE EGEN TABELL
ORLD
LD C85_IND_VST80_K1  ; Z
AND=(300) C85_TYPE_VASK &1  ; VALG AV VASK SE EGEN TABELL
ORLD
LD C02_IND_VST80_K1  ; Z
AND=(300) C02_TYPE_VASK &1  ; VALG AV VASK SE EGEN TABELL
ORLD
LD C82_IND_VST80_K1  ; Z
AND=(300) C82_TYPE_VASK &1  ; VALG AV VASK SE EGEN TABELL
ORLD
LD C31_IND_VST80_K1  ; Z
AND=(300) C31_TYPE_VASK &1  ; VALG AV VASK SE EGEN TABELL
ORLD
ANDLD
ANDNOT K1_VASK_INNE
SET K1_FORSK_LUT_DES  ; FORSKYLLING- LUT-DESINFEKSJON

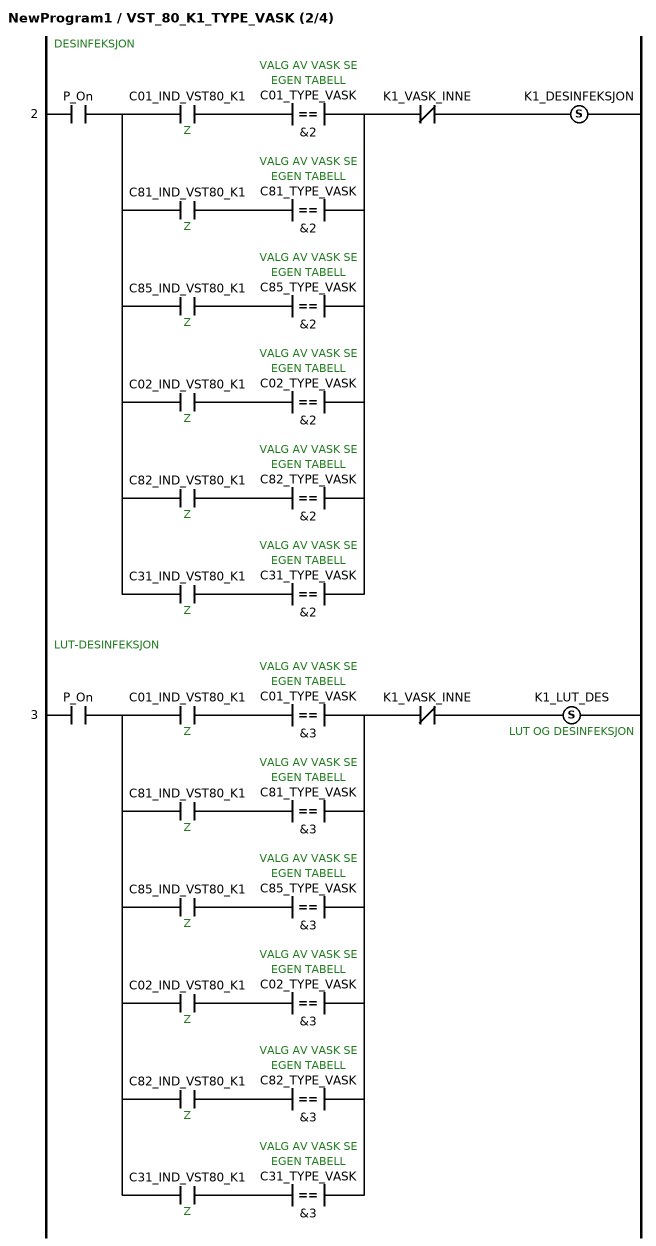
; rung 2: DESINFEKSJON
LD P_On
LD C01_IND_VST80_K1  ; Z
AND=(300) C01_TYPE_VASK &2  ; VALG AV VASK SE EGEN TABELL
LD C81_IND_VST80_K1  ; Z
AND=(300) C81_TYPE_VASK &2  ; VALG AV VASK SE EGEN TABELL
ORLD
LD C85_IND_VST80_K1  ; Z
AND=(300) C85_TYPE_VASK &2  ; VALG AV VASK SE EGEN TABELL
ORLD
LD C02_IND_VST80_K1  ; Z
AND=(300) C02_TYPE_VASK &2  ; VALG AV VASK SE EGEN TABELL
ORLD
LD C82_IND_VST80_K1  ; Z
AND=(300) C82_TYPE_VASK &2  ; VALG AV VASK SE EGEN TABELL
ORLD
LD C31_IND_VST80_K1  ; Z
AND=(300) C31_TYPE_VASK &2  ; VALG AV VASK SE EGEN TABELL
ORLD
ANDLD
ANDNOT K1_VASK_INNE
SET K1_DESINFEKSJON
; rung 3: LUT-DESINFEKSJON
LD P_On
LD C01_IND_VST80_K1  ; Z
AND=(300) C01_TYPE_VASK &3  ; VALG AV VASK SE EGEN TABELL
LD C81_IND_VST80_K1  ; Z
AND=(300) C81_TYPE_VASK &3  ; VALG AV VASK SE EGEN TABELL
ORLD
LD C85_IND_VST80_K1  ; Z
AND=(300) C85_TYPE_VASK &3  ; VALG AV VASK SE EGEN TABELL
ORLD
LD C02_IND_VST80_K1  ; Z
AND=(300) C02_TYPE_VASK &3  ; VALG AV VASK SE EGEN TABELL
ORLD
LD C82_IND_VST80_K1  ; Z
AND=(300) C82_TYPE_VASK &3  ; VALG AV VASK SE EGEN TABELL
ORLD
LD C31_IND_VST80_K1  ; Z
AND=(300) C31_TYPE_VASK &3  ; VALG AV VASK SE EGEN TABELL
ORLD
ANDLD
ANDNOT K1_VASK_INNE
SET K1_LUT_DES  ; LUT OG DESINFEKSJON

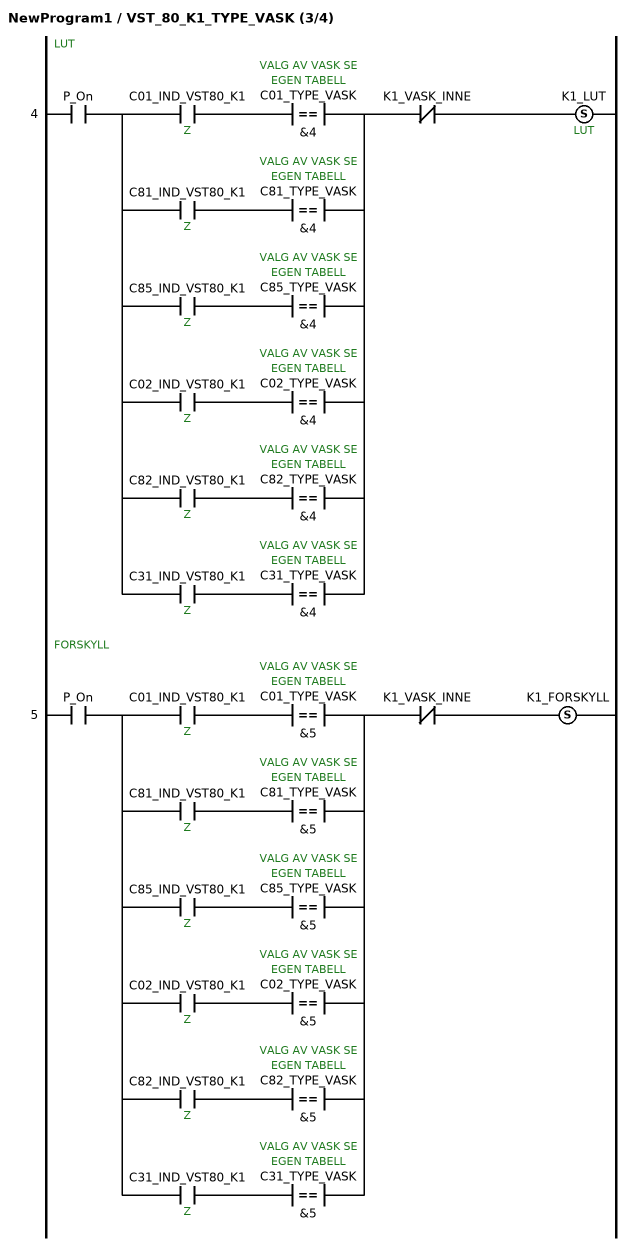
; rung 4: LUT
LD P_On
LD C01_IND_VST80_K1  ; Z
AND=(300) C01_TYPE_VASK &4  ; VALG AV VASK SE EGEN TABELL
LD C81_IND_VST80_K1  ; Z
AND=(300) C81_TYPE_VASK &4  ; VALG AV VASK SE EGEN TABELL
ORLD
LD C85_IND_VST80_K1  ; Z
AND=(300) C85_TYPE_VASK &4  ; VALG AV VASK SE EGEN TABELL
ORLD
LD C02_IND_VST80_K1  ; Z
AND=(300) C02_TYPE_VASK &4  ; VALG AV VASK SE EGEN TABELL
ORLD
LD C82_IND_VST80_K1  ; Z
AND=(300) C82_TYPE_VASK &4  ; VALG AV VASK SE EGEN TABELL
ORLD
LD C31_IND_VST80_K1  ; Z
AND=(300) C31_TYPE_VASK &4  ; VALG AV VASK SE EGEN TABELL
ORLD
ANDLD
ANDNOT K1_VASK_INNE
SET K1_LUT  ; LUT
; rung 5: FORSKYLL
LD P_On
LD C01_IND_VST80_K1  ; Z
AND=(300) C01_TYPE_VASK &5  ; VALG AV VASK SE EGEN TABELL
LD C81_IND_VST80_K1  ; Z
AND=(300) C81_TYPE_VASK &5  ; VALG AV VASK SE EGEN TABELL
ORLD
LD C85_IND_VST80_K1  ; Z
AND=(300) C85_TYPE_VASK &5  ; VALG AV VASK SE EGEN TABELL
ORLD
LD C02_IND_VST80_K1  ; Z
AND=(300) C02_TYPE_VASK &5  ; VALG AV VASK SE EGEN TABELL
ORLD
LD C82_IND_VST80_K1  ; Z
AND=(300) C82_TYPE_VASK &5  ; VALG AV VASK SE EGEN TABELL
ORLD
LD C31_IND_VST80_K1  ; Z
AND=(300) C31_TYPE_VASK &5  ; VALG AV VASK SE EGEN TABELL
ORLD
ANDLD
ANDNOT K1_VASK_INNE
SET K1_FORSKYLL

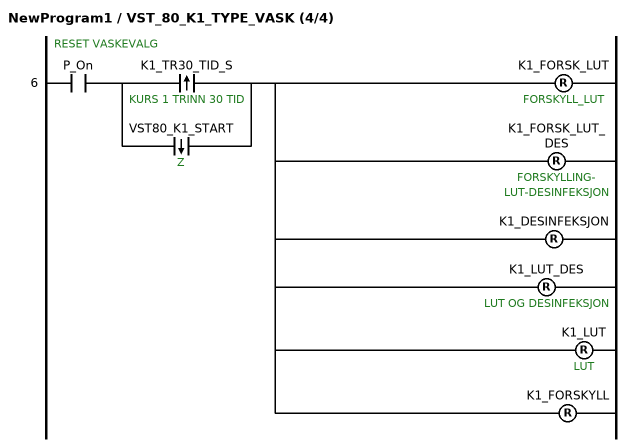
; rung 6: RESET VASKEVALG
LD P_On
@LD K1_TR30_TID_S  ; KURS 1 TRINN 30 TID
%OR VST80_K1_START  ; Z
ANDLD
RSET K1_FORSK_LUT  ; FORSKYLL_LUT
RSET K1_FORSK_LUT_DES  ; FORSKYLLING- LUT-DESINFEKSJON
RSET K1_DESINFEKSJON
RSET K1_LUT_DES  ; LUT OG DESINFEKSJON
RSET K1_LUT  ; LUT
RSET K1_FORSKYLL

### Section VST80_K1_DR_STATUS

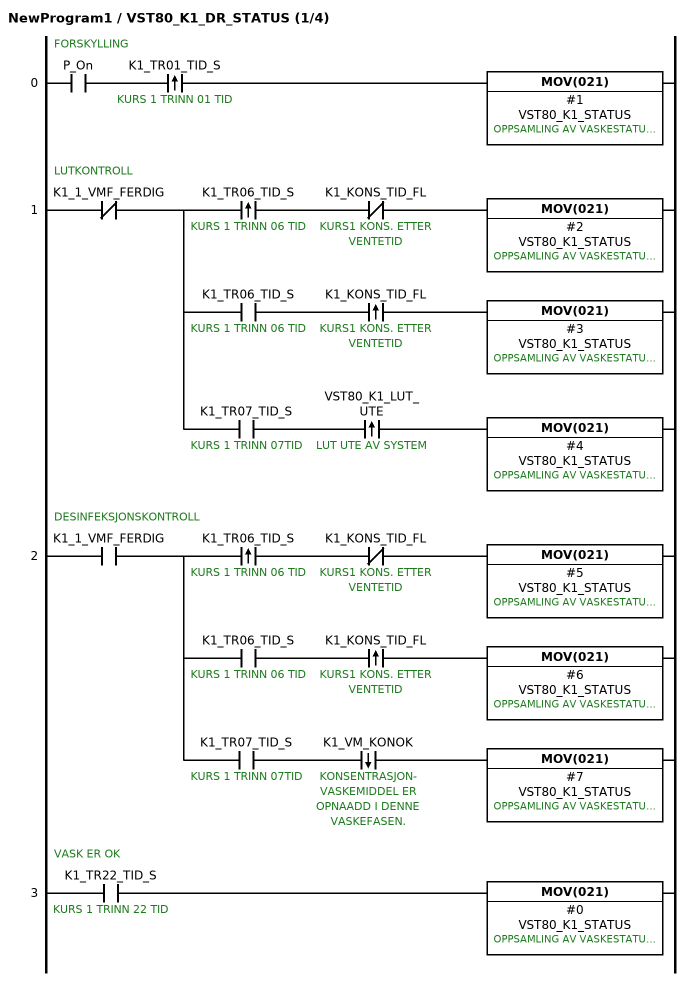
; rung 0: FORSKYLLING
LD P_On
@AND K1_TR01_TID_S  ; KURS 1 TRINN 01 TID
MOV(021) #1 VST80_K1_STATUS  ; OPPSAMLING AV VASKESTATUS UNDER VASK
; rung 1: LUTKONTROLL
LDNOT K1_1_VMF_FERDIG
OUT TR0
@AND K1_TR06_TID_S  ; KURS 1 TRINN 06 TID
ANDNOT K1_KONS_TID_FL  ; KURS1 KONS. ETTER VENTETID
MOV(021) #2 VST80_K1_STATUS  ; OPPSAMLING AV VASKESTATUS UNDER VASK
LD TR0
AND K1_TR06_TID_S  ; KURS 1 TRINN 06 TID
@AND K1_KONS_TID_FL  ; KURS1 KONS. ETTER VENTETID
MOV(021) #3 VST80_K1_STATUS  ; OPPSAMLING AV VASKESTATUS UNDER VASK
LD TR0
AND K1_TR07_TID_S  ; KURS 1 TRINN 07TID
@AND VST80_K1_LUT_UTE  ; LUT UTE AV SYSTEM
MOV(021) #4 VST80_K1_STATUS  ; OPPSAMLING AV VASKESTATUS UNDER VASK
; rung 2: DESINFEKSJONSKONTROLL
LD K1_1_VMF_FERDIG
OUT TR0
@AND K1_TR06_TID_S  ; KURS 1 TRINN 06 TID
ANDNOT K1_KONS_TID_FL  ; KURS1 KONS. ETTER VENTETID
MOV(021) #5 VST80_K1_STATUS  ; OPPSAMLING AV VASKESTATUS UNDER VASK
LD TR0
AND K1_TR06_TID_S  ; KURS 1 TRINN 06 TID
@AND K1_KONS_TID_FL  ; KURS1 KONS. ETTER VENTETID
MOV(021) #6 VST80_K1_STATUS  ; OPPSAMLING AV VASKESTATUS UNDER VASK
LD TR0
AND K1_TR07_TID_S  ; KURS 1 TRINN 07TID
%AND K1_VM_KONOK  ; KONSENTRASJON-VASKEMIDDEL ER OPNAADD I DENNE VASKEFASEN.
MOV(021) #7 VST80_K1_STATUS  ; OPPSAMLING AV VASKESTATUS UNDER VASK
; rung 3: VASK ER OK
LD K1_TR22_TID_S  ; KURS 1 TRINN 22 TID
MOV(021) #0 VST80_K1_STATUS  ; OPPSAMLING AV VASKESTATUS UNDER VASK

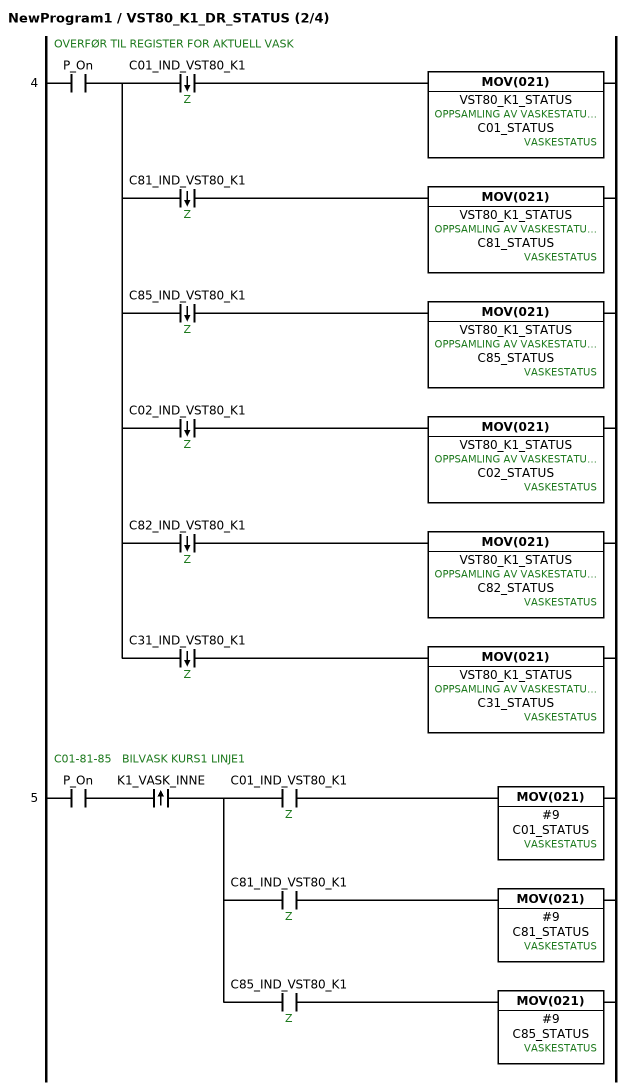
; rung 4: OVERFØR TIL REGISTER FOR AKTUELL VASK
LD P_On
OUT TR0
%AND C01_IND_VST80_K1  ; Z
MOV(021) VST80_K1_STATUS C01_STATUS  ; OPPSAMLING AV VASKESTATUS UNDER VASK, VASKESTATUS
LD TR0
%AND C81_IND_VST80_K1  ; Z
MOV(021) VST80_K1_STATUS C81_STATUS  ; OPPSAMLING AV VASKESTATUS UNDER VASK, VASKESTATUS
LD TR0
%AND C85_IND_VST80_K1  ; Z
MOV(021) VST80_K1_STATUS C85_STATUS  ; OPPSAMLING AV VASKESTATUS UNDER VASK, VASKESTATUS
LD TR0
%AND C02_IND_VST80_K1  ; Z
MOV(021) VST80_K1_STATUS C02_STATUS  ; OPPSAMLING AV VASKESTATUS UNDER VASK, VASKESTATUS
LD TR0
%AND C82_IND_VST80_K1  ; Z
MOV(021) VST80_K1_STATUS C82_STATUS  ; OPPSAMLING AV VASKESTATUS UNDER VASK, VASKESTATUS
LD TR0
%AND C31_IND_VST80_K1  ; Z
MOV(021) VST80_K1_STATUS C31_STATUS  ; OPPSAMLING AV VASKESTATUS UNDER VASK, VASKESTATUS
; rung 5: C01-81-85   BILVASK KURS1 LINJE1
LD P_On
@AND K1_VASK_INNE
OUT TR0
AND C01_IND_VST80_K1  ; Z
MOV(021) #9 C01_STATUS  ; VASKESTATUS
LD TR0
AND C81_IND_VST80_K1  ; Z
MOV(021) #9 C81_STATUS  ; VASKESTATUS
LD TR0
AND C85_IND_VST80_K1  ; Z
MOV(021) #9 C85_STATUS  ; VASKESTATUS

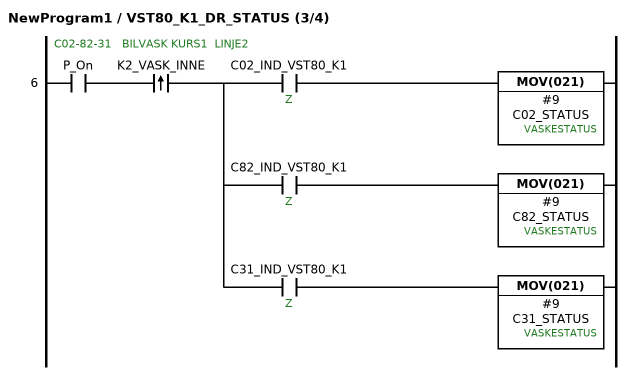
; rung 6: C02-82-31   BILVASK KURS1  LINJE2
LD P_On
@AND K2_VASK_INNE
OUT TR0
AND C02_IND_VST80_K1  ; Z
MOV(021) #9 C02_STATUS  ; VASKESTATUS
LD TR0
AND C82_IND_VST80_K1  ; Z
MOV(021) #9 C82_STATUS  ; VASKESTATUS
LD TR0
AND C31_IND_VST80_K1  ; Z
MOV(021) #9 C31_STATUS  ; VASKESTATUS

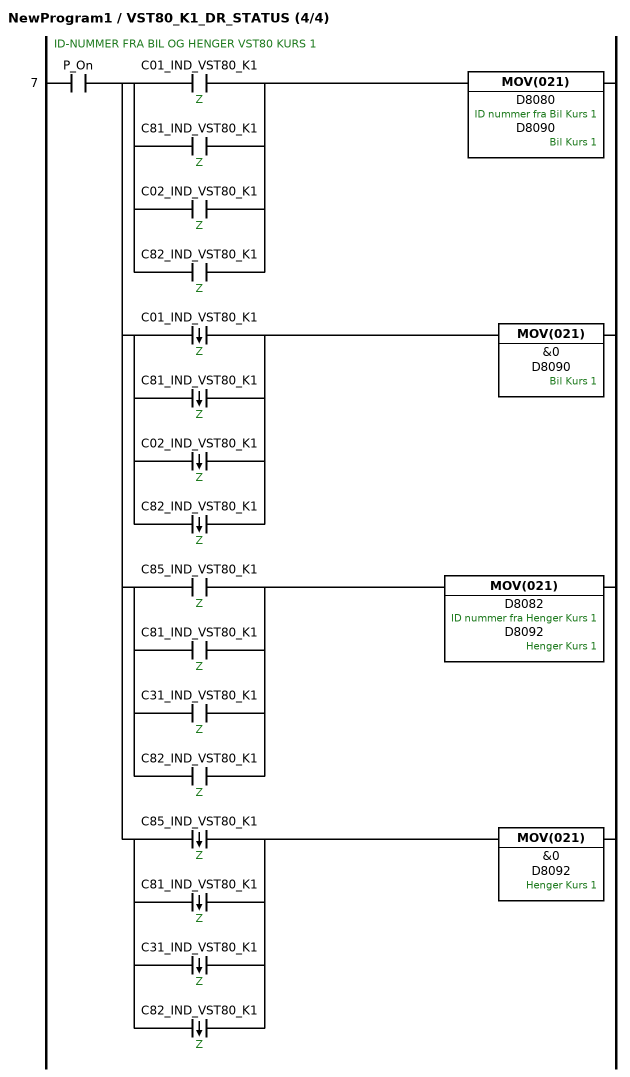
; rung 7: ID-NUMMER FRA BIL OG HENGER VST80 KURS 1
LD P_On
OUT TR0
LD C01_IND_VST80_K1  ; Z
OR C81_IND_VST80_K1  ; Z
OR C02_IND_VST80_K1  ; Z
OR C82_IND_VST80_K1  ; Z
ANDLD
MOV(021) D8080 D8090  ; ID nummer fra Bil Kurs 1, Bil Kurs 1
LD TR0
%LD C01_IND_VST80_K1  ; Z
%OR C81_IND_VST80_K1  ; Z
%OR C02_IND_VST80_K1  ; Z
%OR C82_IND_VST80_K1  ; Z
ANDLD
MOV(021) &0 D8090  ; Bil Kurs 1
LD TR0
LD C85_IND_VST80_K1  ; Z
OR C81_IND_VST80_K1  ; Z
OR C31_IND_VST80_K1  ; Z
OR C82_IND_VST80_K1  ; Z
ANDLD
MOV(021) D8082 D8092  ; ID nummer fra Henger Kurs 1, Henger Kurs 1
LD TR0
%LD C85_IND_VST80_K1  ; Z
%OR C81_IND_VST80_K1  ; Z
%OR C31_IND_VST80_K1  ; Z
%OR C82_IND_VST80_K1  ; Z
ANDLD
MOV(021) &0 D8092  ; Henger Kurs 1

### Section VST80_K1_FUNKSJON
; Dette programmet styrer kommandoene til vaskestasjonen.

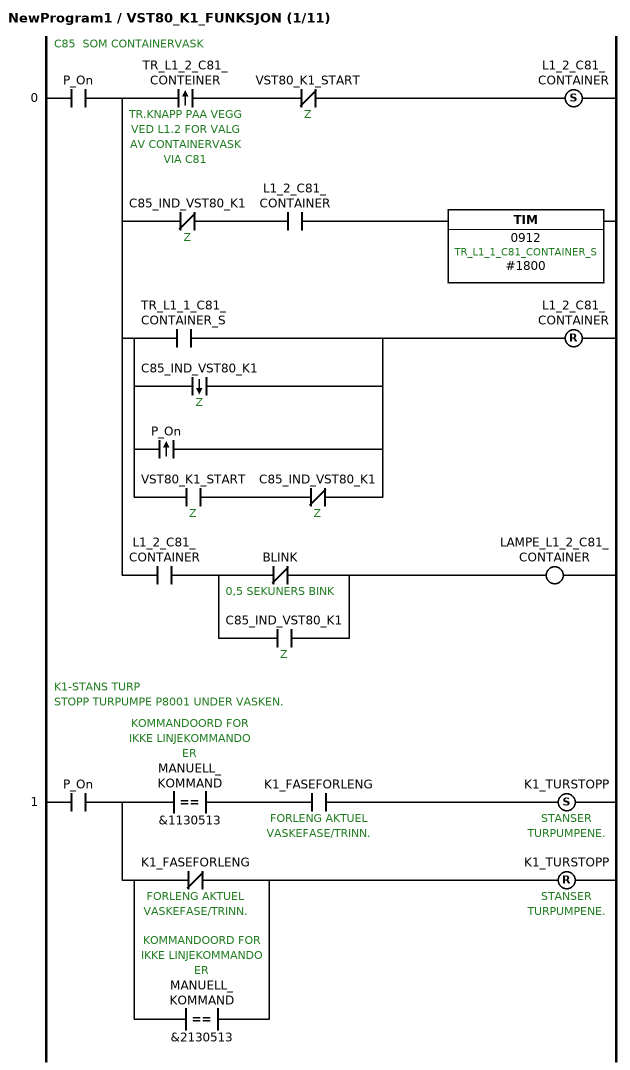
; rung 0: C85  SOM CONTAINERVASK
LD P_On
OUT TR0
@AND TR_L1_2_C81_CONTEINER  ; TR.KNAPP PAA VEGG VED L1.2 FOR VALG AV CONTAINERVASK VIA C81
ANDNOT VST80_K1_START  ; Z
SET L1_2_C81_CONTAINER
LD TR0
ANDNOT C85_IND_VST80_K1  ; Z
AND L1_2_C81_CONTAINER
TIM 0912 #1800  ; TR_L1_1_C81_CONTAINER_S
LD TR0
LD TR_L1_1_C81_CONTAINER_S
%OR C85_IND_VST80_K1  ; Z
@OR P_On
LD VST80_K1_START  ; Z
ANDNOT C85_IND_VST80_K1  ; Z
ORLD
ANDLD
RSET L1_2_C81_CONTAINER
LD TR0
AND L1_2_C81_CONTAINER
LDNOT BLINK  ; 0,5 SEKUNERS BINK
OR C85_IND_VST80_K1  ; Z
ANDLD
OUT LAMPE_L1_2_C81_CONTAINER
; rung 1: K1-STANS TURP / STOPP TURPUMPE P8001 UNDER VASKEN.
LD P_On
OUT TR0
AND=L(301) MANUELL_KOMMAND &1130513  ; KOMMANDOORD FOR IKKE LINJEKOMMANDOER
AND K1_FASEFORLENG  ; FORLENG AKTUEL VASKEFASE/TRINN.
SET K1_TURSTOPP  ; STANSER TURPUMPENE.
LD TR0
LDNOT K1_FASEFORLENG  ; FORLENG AKTUEL VASKEFASE/TRINN.
OR=L(301) MANUELL_KOMMAND &2130513  ; KOMMANDOORD FOR IKKE LINJEKOMMANDOER
ANDLD
RSET K1_TURSTOPP  ; STANSER TURPUMPENE.

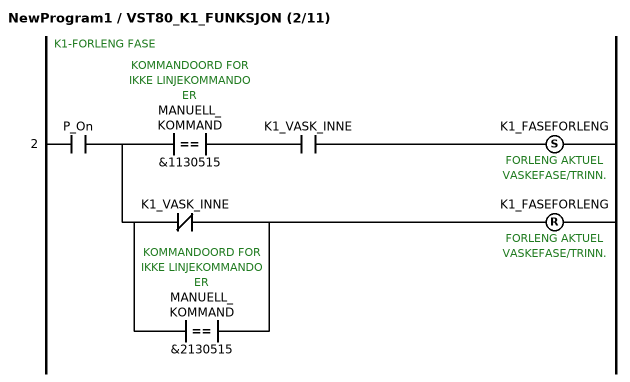
; rung 2: K1-FORLENG FASE
LD P_On
OUT TR0
AND=L(301) MANUELL_KOMMAND &1130515  ; KOMMANDOORD FOR IKKE LINJEKOMMANDOER
AND K1_VASK_INNE
SET K1_FASEFORLENG  ; FORLENG AKTUEL VASKEFASE/TRINN.
LD TR0
LDNOT K1_VASK_INNE
OR=L(301) MANUELL_KOMMAND &2130515  ; KOMMANDOORD FOR IKKE LINJEKOMMANDOER
ANDLD
RSET K1_FASEFORLENG  ; FORLENG AKTUEL VASKEFASE/TRINN.

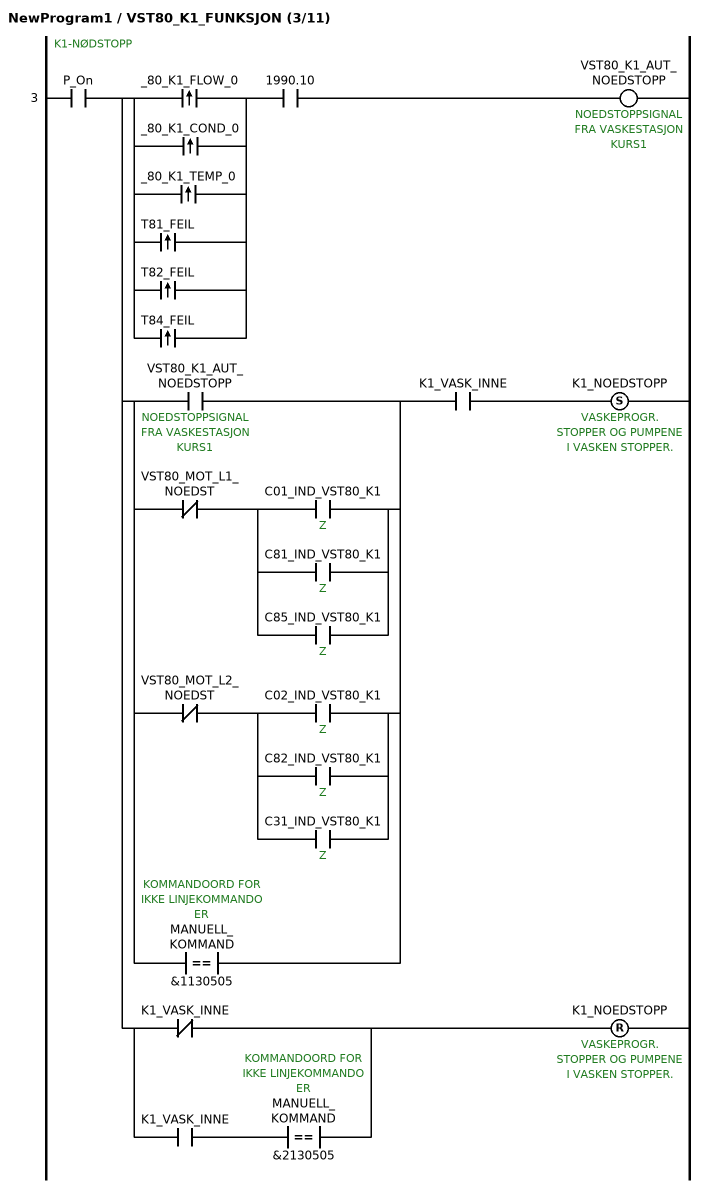
; rung 3: K1-NØDSTOPP
LD P_On
OUT TR0
@LD _80_K1_FLOW_0
@OR _80_K1_COND_0
@OR _80_K1_TEMP_0
@OR T81_FEIL
@OR T82_FEIL
@OR T84_FEIL
ANDLD
AND 1990.10
OUT VST80_K1_AUT_NOEDSTOPP  ; NOEDSTOPPSIGNAL FRA VASKESTASJON KURS1
LD TR0
LD VST80_K1_AUT_NOEDSTOPP  ; NOEDSTOPPSIGNAL FRA VASKESTASJON KURS1
LDNOT VST80_MOT_L1_NOEDST
LD C01_IND_VST80_K1  ; Z
OR C81_IND_VST80_K1  ; Z
OR C85_IND_VST80_K1  ; Z
ANDLD
ORLD
LDNOT VST80_MOT_L2_NOEDST
LD C02_IND_VST80_K1  ; Z
OR C82_IND_VST80_K1  ; Z
OR C31_IND_VST80_K1  ; Z
ANDLD
ORLD
OR=L(301) MANUELL_KOMMAND &1130505  ; KOMMANDOORD FOR IKKE LINJEKOMMANDOER
ANDLD
AND K1_VASK_INNE
SET K1_NOEDSTOPP  ; VASKEPROGR. STOPPER OG PUMPENE I VASKEN STOPPER.
LD TR0
LDNOT K1_VASK_INNE
LD K1_VASK_INNE
AND=L(301) MANUELL_KOMMAND &2130505  ; KOMMANDOORD FOR IKKE LINJEKOMMANDOER
ORLD
ANDLD
RSET K1_NOEDSTOPP  ; VASKEPROGR. STOPPER OG PUMPENE I VASKEN STOPPER.

